TYPE "UDT_ZC_DISP_PPAL_TOT"
VERSION : 0.1
   STRUCT
      Orden : Bool;   // Orden activacion
      ResetProceso : Bool;   // Orden reset proceso
      ResetParcial : Bool;   // Orden reset parcial
      ResetTotal : Bool;   // Orden reset total
      ValorProceso : LReal;   // Valor actual proceso
      ValorParcial : LReal;   // Valor actual parcial
      ValorTotal : LReal;   // Valor actual total
   END_STRUCT;

END_TYPE

